TYPE ST_GantryXY :
    STRUCT
        Length              : LREAL;
        LeftAxis            : ST_AxisRecipe;
        RightAxis           : ST_AxisRecipe;
        CylinderExtendTime : LREAL;
        CylinderRetractTime : LREAL;
    END_STRUCT
END_TYPE

(* stored: Version 1.1.0.1
   DUT ST_GantryXY: Id {0c91b655-e341-4901-a4e8-51cfd7b8e196} *)
